FUNCTION_BLOCK AX_OR_3 (* FB to calculate boolean OR *)
  (* Standard: 61499-2 *)
  (* Version 1.0, 2024-10-23, franz *)
  PACKAGE io::adp::boolean;
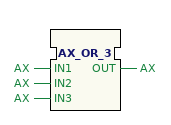
  SOCKETS
    IN1 : AX; (* OR input 1 *)
    IN2 : AX; (* OR input 2 *)
    IN3 : AX; (* OR input 3 *)
  END_SOCKETS
  PLUGS
    OUT : AX; (* OR result *)
  END_PLUGS
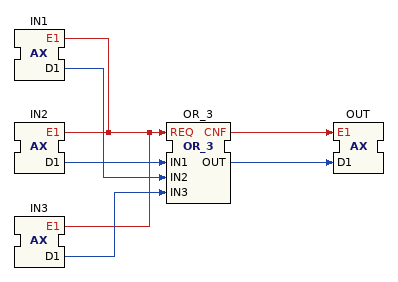
  FBS
    OR_3 : OR_3;
  END_FBS
  EVENT_CONNECTIONS
    IN1.E1 TO OR_3.REQ;
    IN2.E1 TO OR_3.REQ;
    OR_3.CNF TO OUT.E1;
    IN3.E1 TO OR_3.REQ;
  END_CONNECTIONS
  DATA_CONNECTIONS
    IN1.D1 TO OR_3.IN1;
    IN2.D1 TO OR_3.IN2;
    OR_3.OUT TO OUT.D1;
    IN3.D1 TO OR_3.IN3;
  END_CONNECTIONS
END_FUNCTION_BLOCK
